FUNCTION_BLOCK AxisCtrl
VAR_INPUT
END_VAR
VAR_OUTPUT
END_VAR
VAR
	axis : AXIS_REF;
	state : Stage_t;
	
	moveAbs: MC_MoveAbsolute;
	moveAbsOut: ST_McOutputs;

	moveAbs2: MC_MoveAbsolute;
	moveAbsOut2: ST_McOutputs;
	
	power: MC_Power;
	powerOut : ST_McOutputs;
	
	reset: MC_Reset;
	resetOut : ST_McOutputs;
	
	halt: MC_Halt;
	haltOut : ST_McOutputs;
	
	cmd_pos : LREAL;
	cmd_vel : LREAL;
	cmd_acc : LREAL;
	cmd_vel_end : LREAL;
	cmd_need_exe : BOOL;
	cmd_need_home : BOOL := TRUE;
	cmd_halt : BOOL := FALSE;
	
	readActPos: MC_ReadActualPosition;
	readActVel: MC_ReadActualVelocity;
	
	actPosOut : ST_McOutputs;
	actVelOut : ST_McOutputs;
	
	actual_pos : LREAL;
	actual_vel : LREAL;
	
	(* Festo Homing*)
	homeFesto: Festo_MC_Home;
	homeFestoOut : ST_McOutputs;
	
	amsAddr AT %I* : AMSADDR;
	deviceNetID	:T_AmsNetId	:= '192.168.2.43.2.1';
	
	driveError: Festo_GetDriveError;
	
	// variables for function block "Festo_GetDriveError"
	GetErrorEnable		:BOOL;
	GetErrorBusy		:BOOL;
	DriveInErrorState	:BOOL;
	DriveErrorNumber	:ARRAY [1..4] OF DWORD;
	GetErrorWasAbortive	:BOOL;
	GetErrorId	: UDINT;

	error : BOOL := FALSE;
	resetTest : BOOL := FALSE;
	enableTest : BOOL := FALSE;
	recovered : BOOL := FALSE;
	afterHomeTimer : TON;
END_VAR


axis.ReadStatus();

power.Enable := TRUE;
IF powerOut.Done THEN
	homeFesto.Execute := TRUE;
END_IF


IF homeFestoOut.Done OR (axis.Status.Error AND axis.Status.ErrorID = 18000) THEN
	afterHomeTimer(IN:=TRUE, PT:=T#500MS);
	IF afterHomeTimer.Q THEN
		reset.Execute := TRUE;
	END_IF
END_IF

ActPower();
ActRead();
ActHalt();
actMove();
ActReset();
ActHomeFesto();

ACTION ActHalt:
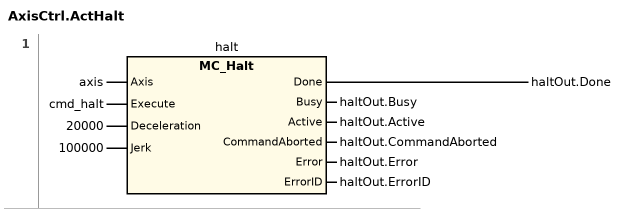
// NETWORK 1
halt(
    Axis := axis,
    Execute := cmd_halt,
    Deceleration := 20000,
    Jerk := 100000,
    Busy => haltOut.Busy,
    Active => haltOut.Active,
    CommandAborted => haltOut.CommandAborted,
    Error => haltOut.Error,
    ErrorID => haltOut.ErrorID); // MC_Halt
haltOut.Done := halt.Done;
END_ACTION

ACTION ActHomeFesto:
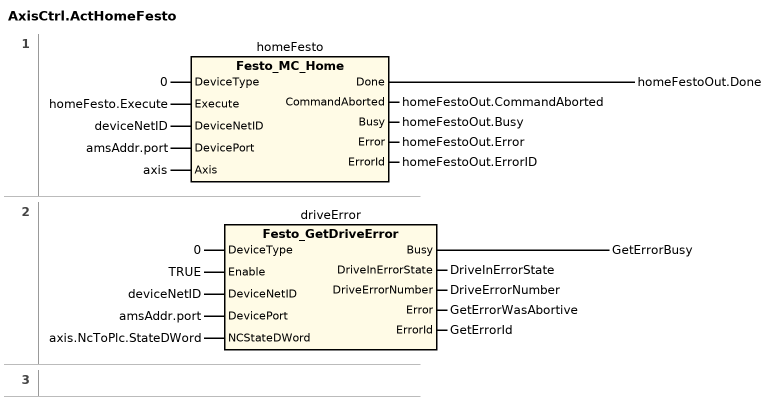
// NETWORK 1
homeFesto(
    DeviceType := 0,
    Execute := homeFesto.Execute,
    DeviceNetID := deviceNetID,
    DevicePort := amsAddr.port,
    Axis := axis,
    CommandAborted => homeFestoOut.CommandAborted,
    Busy => homeFestoOut.Busy,
    Error => homeFestoOut.Error,
    ErrorId => homeFestoOut.ErrorID); // Festo_MC_Home
homeFestoOut.Done := homeFesto.Done;

// NETWORK 2
driveError(
    DeviceType := 0,
    Enable := TRUE,
    DeviceNetID := deviceNetID,
    DevicePort := amsAddr.port,
    NCStateDWord := axis.NcToPlc.StateDWord,
    DriveInErrorState => DriveInErrorState,
    DriveErrorNumber => DriveErrorNumber,
    Error => GetErrorWasAbortive,
    ErrorId => GetErrorId); // Festo_GetDriveError
GetErrorBusy := driveError.Busy;

// NETWORK 3
END_ACTION

ACTION ActMove:
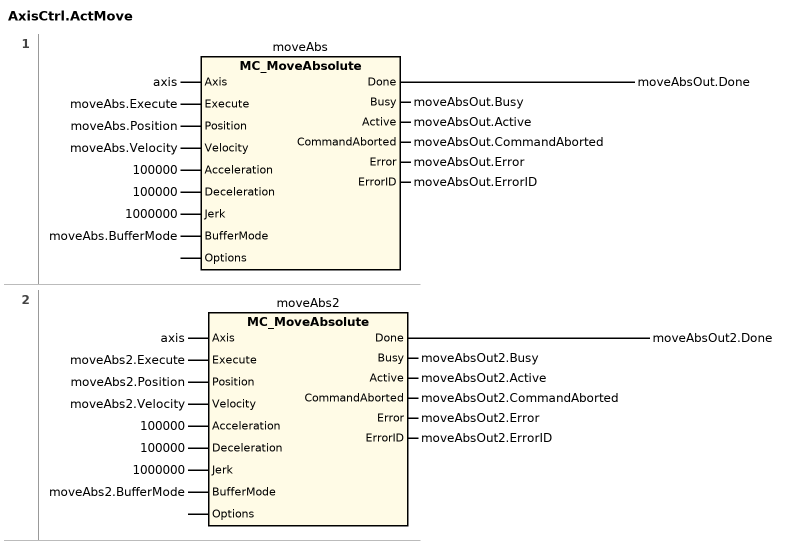
// NETWORK 1
moveAbs(
    Axis := axis,
    Execute := moveAbs.Execute,
    Position := moveAbs.Position,
    Velocity := moveAbs.Velocity,
    Acceleration := 100000,
    Deceleration := 100000,
    Jerk := 1000000,
    BufferMode := moveAbs.BufferMode,
    Busy => moveAbsOut.Busy,
    Active => moveAbsOut.Active,
    CommandAborted => moveAbsOut.CommandAborted,
    Error => moveAbsOut.Error,
    ErrorID => moveAbsOut.ErrorID); // MC_MoveAbsolute
moveAbsOut.Done := moveAbs.Done;

// NETWORK 2
moveAbs2(
    Axis := axis,
    Execute := moveAbs2.Execute,
    Position := moveAbs2.Position,
    Velocity := moveAbs2.Velocity,
    Acceleration := 100000,
    Deceleration := 100000,
    Jerk := 1000000,
    BufferMode := moveAbs2.BufferMode,
    Busy => moveAbsOut2.Busy,
    Active => moveAbsOut2.Active,
    CommandAborted => moveAbsOut2.CommandAborted,
    Error => moveAbsOut2.Error,
    ErrorID => moveAbsOut2.ErrorID); // MC_MoveAbsolute
moveAbsOut2.Done := moveAbs2.Done;
END_ACTION

ACTION ActPower:
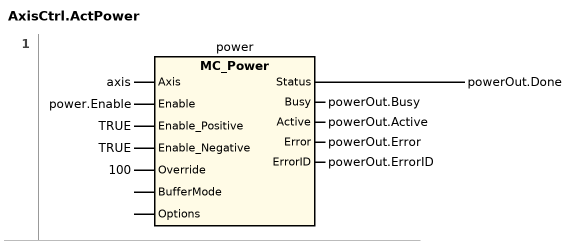
// NETWORK 1
power(
    Axis := axis,
    Enable := power.Enable,
    Enable_Positive := TRUE,
    Enable_Negative := TRUE,
    Override := 100,
    Busy => powerOut.Busy,
    Active => powerOut.Active,
    Error => powerOut.Error,
    ErrorID => powerOut.ErrorID); // MC_Power
powerOut.Done := power.Status;
END_ACTION

ACTION ActRead:
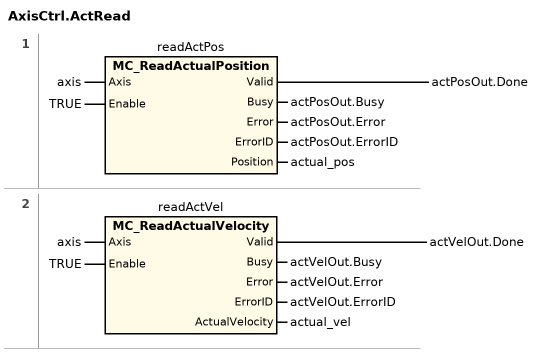
// NETWORK 1
readActPos(
    Axis := axis,
    Enable := TRUE,
    Busy => actPosOut.Busy,
    Error => actPosOut.Error,
    ErrorID => actPosOut.ErrorID,
    Position => actual_pos); // MC_ReadActualPosition
actPosOut.Done := readActPos.Valid;

// NETWORK 2
readActVel(
    Axis := axis,
    Enable := TRUE,
    Busy => actVelOut.Busy,
    Error => actVelOut.Error,
    ErrorID => actVelOut.ErrorID,
    ActualVelocity => actual_vel); // MC_ReadActualVelocity
actVelOut.Done := readActVel.Valid;
END_ACTION

ACTION ActReset:
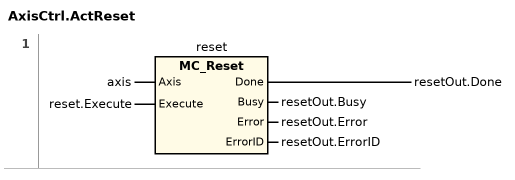
// NETWORK 1
reset(
    Axis := axis,
    Execute := reset.Execute,
    Busy => resetOut.Busy,
    Error => resetOut.Error,
    ErrorID => resetOut.ErrorID); // MC_Reset
resetOut.Done := reset.Done;
END_ACTION

END_FUNCTION_BLOCK

(* stored: Version 1.1.0.1, ProductVersion 3.1.4020.12
   POU AxisCtrl: Id {01aa567d-2819-4b37-ab34-80f23c757336}, SpecialFunc None
   Action ActHalt: Id {d5c01865-609c-415d-9648-2a332c575221}
   Action ActHomeFesto: Id {6d10a84e-e1e9-4b9b-8461-9dd3fb3dcc22}
   Action ActMove: Id {247383c3-3462-4c47-9232-c32450d351cb}
   Action ActPower: Id {22a22ddc-1a7b-4ee3-afcd-5be87eff8605}
   Action ActRead: Id {142750ff-8f7d-42cb-81db-ad518e9855c2}
   Action ActReset: Id {64847ba5-ab45-49df-a045-5787b238cbe1} *)
